FUNCTION_BLOCK FuelMeasurement
VAR CONSTANT
	TankVolume : INT := 334; // The volume may vary depending on the tank volume.
	
END_VAR
VAR_INPUT
	bFuelMeasurement : BOOL := TRUE;
	
END_VAR
VAR_OUTPUT
	timeElapsed: TIME := T#0S;
	
	valveN1 : BOOL := FALSE;
	valveN2 : BOOL := FALSE;
	bEndFB : BOOL;
	FuelVolumePerSec : REAL := 0;
	
END_VAR
VAR
	bMeasurementDone : BOOL;
	readyToCount : BOOL := FALSE;
	timeStart: TIME;  
 	timerRunning: BOOL := FALSE;
	
	readyToClose : BOOL := FALSE;
	
	TimeToReal : REAL;
	INT1: INT :=0;
END_VAR

CASE INT1 OF
0:
	IF GVL.sensorN1 AND GVL.sensorN2 THEN
		INT1 := 10;
	END_IF
10:  //Ready
	IF GVL.sensorN1 AND GVL.sensorN2 AND bFuelMeasurement THEN
	valveN1 := TRUE;
	valveN2 := TRUE;
	INT1 := 20;
	END_IF  
20:  //Wait for upper sensor
	IF NOT GVL.sensorN1 THEN
	timeStart := TIME();
	timerRunning := TRUE;
	INT1 := 30;
	END_IF   
30: //Wait for lower sensor
	IF NOT GVL.sensorN2 THEN
	timeElapsed := TIME() - timeStart;
	timerRunning := FALSE;
	
	TimeToReal := (TIME_TO_REAL(timeElapsed)/ 1000); // The unit of TimeToReal is Second.
	FuelVolumePerSec := TankVolume / (TimeToReal/60) ;

	INT1 := 40;
	END_IF
40: //Measurement finished

	valveN1 := FALSE;
	valveN2 := FALSE;
	bEndFB := TRUE;
	IF GVL.sensorN1 AND GVL.sensorN2 THEN
	INT1 := 10;
	END_IF
	
END_CASE;

END_FUNCTION_BLOCK

(* stored: Version 1.1.0.1, ProductVersion 3.1.4024.13
   POU FuelMeasurement: Id {e8713979-005e-49c2-8c38-3baad67b76ee}, SpecialFunc None *)
